// Type alias for a single wide character string.
TYPE T_WChar : WSTRING(1); END_TYPE

(* stored: Version 1.1.0.1
   DUT T_WChar: Id {26546536-84ed-01ee-3d87-ed30002f9cf2} *)
